# B&R Automation Studio project NAINV104C00R8L515F00 (part 22)

#### Local.var
```iecst
(*2019-06-17*)
(**)
(*Local Action, State & Status*)
VAR
	eAct : eConvAction := ConvActIdle;
	eStat : eConvAction := ConvActIdle;
	eStatus : eFBStatus := Idle;
	udiStatus : UDINT := 0;
	sStatTxt : STRING[200] := '';
	a_sStatText : ARRAY[0..60] OF STRING[200] := ['Idling','Initializing','Initializing With Reverse','Initializing With Pusher','Initializing With Puller','Initializing With Reject','Initializing With Inspection','Entering Board','Entering Board Until Inlet Signal Off','Entering Board With Reverse','Reversing Board','Reversing Board With Immediate Start Conv','Entering Board With Puller','Entering Board With Reject','Entering Board With Inspection','Pre Exiting Board','Resuming Reject Board',2('Exiting Board'),2('Exiting Board With Pusher'),'Pusher Setting All Control','Pusher Resetting All Control','Pusher Setting Extend','Pusher Setting Retract','Pusher Extending','Pusher Retracting','Puller Setting All Control','Puller Resetting All Control','Puller Setting Extend','Puller Setting Retract','Puller Extending','Puller Retracting','Rotating Setting All Control','Rotating Resetting All Control','Rotating Setting Home','Rotating Setting Remote','Rotating Turning Home','Rotating Turning Remote','Reject Setting All Control','Reject Resetting All Control','Reject Setting Up','Reject Setting Down','Reject Going Up','Reject Going Down','Stopping','Stopping With Pusher','Stopping With Puller','Stopping With Reject','Turning On Motor Signal','Turning On Motor Direction','Turning Off Motor Signal','Turning Off Motor Direction','Turning On All Motor Output','Turning Off All Motor Output',6('')];
END_VAR
(**)
(*Local Alarm*)
VAR
	tyAlmData : tyAlmDat;
	a_tyAlmText : ARRAY[10000..10199] OF tyAlmTxt := [(sAlmText:='Multi Board Detected While Conveyor Initial',sRcyText:='Operation Interrupted By Multiple Board. Remove Extra Boards And Resume Operation.'),(sAlmText:='Board Not Present At Outlet Sensor (L - R) While Conveyor Initial',sRcyText:='Operation Interrupted By Jam Board. Remove The Jam Board To Resume Operation.'),(sAlmText:='Board Not Present At Outlet Sensor (R - L) While Conveyor Initial',sRcyText:='Operation Interrupted By Jam Board. Remove The Jam Board To Resume Operation.'),(sAlmText:='Multi Board Detected While Conveyor Initial With Reverse',sRcyText:='Operation Interrupted By Multiple Board. Remove Extra Boards And Resume Operation.'),(sAlmText:='Board Not Present At Outlet Sensor (L - R) While Conveyor Initial With Reverse',sRcyText:='Operation Interrupted By Jam Board. Remove The Jam Board To Resume Operation.'),(sAlmText:='Board Not Present At Outlet Sensor (R - L) While Conveyor Initial With Reverse',sRcyText:='Operation Interrupted By Jam Board. Remove The Jam Board To Resume Operation.'),(sAlmText:='Pusher Extend Sensor Off Time Out In Retract Check While Conveyor Initial With Pusher',sRcyText:='Sensor Timeout Expired Before Operation Completed. Sensor Operation Is Abnormal. Solve The Error To Resume Operation.'),(sAlmText:='Pusher Retract Sensor On Time Out In Retract Check While Conveyor Initial With Pusher',sRcyText:='Sensor Timeout Expired Before Operation Completed. Sensor Operation Is Abnormal. Solve The Error To Resume Operation.'),(sAlmText:='Pusher Retract Safety Sensor Error In Retract Check While Conveyor Initial With Pusher',sRcyText:='Safety System Has Been Triggered. All Operations Are Disable. Remove the Obstacle That Triggered The Safety Interlock To Resume Operation.'),(sAlmText:='Multi Board Detected While Conveyor Initial With Pusher',sRcyText:='Operation Interrupted By Multiple Board. Remove Extra Boards And Resume Operation.'),(sAlmText:='Board Not Present At Outlet Sensor (L - R) While Conveyor Initial With Pusher',sRcyText:='Operation Interrupted By Jam Board. Remove The Jam Board To Resume Operation.'),(sAlmText:='Board Not Present At Outlet Sensor (R - L) While Conveyor Initial With Pusher',sRcyText:='Operation Interrupted By Jam Board. Remove The Jam Board To Resume Operation.'),(sAlmText:='Rotator Home Sensor On Time Out In Home Check While Conveyor Initial With Puller',sRcyText:='Sensor Timeout Expired Before Operation Completed. Sensor Operation Is Abnormal. Solve The Error To Resume Operation.'),(sAlmText:='Rotator Remote Sensor Off Time Out In Home Check While Conveyor Initial With Puller',sRcyText:='Sensor Timeout Expired Before Operation Completed. Sensor Operation Is Abnormal. Solve The Error To Resume Operation.'),(sAlmText:='Rotator Home Safety Sensor Error In Home Check While Conveyor Initial With Puller',sRcyText:='Safety System Has Been Triggered. All Operations Are Disable. Remove the Obstacle That Triggered The Safety Interlock To Resume Operation.'),(sAlmText:='Puller Extend Sensor Off Time Out In Retract Check While Conveyor Initial With Puller',sRcyText:='Sensor Timeout Expired Before Operation Completed. Sensor Operation Is Abnormal. Solve The Error To Resume Operation.'),(sAlmText:='Puller Retract Sensor On Time Out In Retract Check While Conveyor Initial With Puller',sRcyText:='Sensor Timeout Expired Before Operation Completed. Sensor Operation Is Abnormal. Solve The Error To Resume Operation.'),(sAlmText:='Puller Retract Safety Sensor Error In Retract Check While Conveyor Initial With Puller',sRcyText:='Safety System Has Been Triggered. All Operations Are Disable. Remove the Obstacle That Triggered The Safety Interlock To Resume Operation.'),(sAlmText:='Multi Board Detected While Conveyor Initial With Puller',sRcyText:='Operation Interrupted By Multiple Board. Remove Extra Boards And Resume Operation.'),(sAlmText:='Board Not Present At Outlet Sensor (L - R) While Conveyor Initial With Puller',sRcyText:='Operation Interrupted By Jam Board. Remove The Jam Board To Resume Operation.'),(sAlmText:='Board Not Present At Outlet Sensor (R - L) While Conveyor Initial With Puller',sRcyText:='Operation Interrupted By Jam Board. Remove The Jam Board To Resume Operation.'),(sAlmText:='Multi Board Detected While Conveyor Enter Board',sRcyText:='Operation Interrupted By Multiple Board. Remove Extra Boards And Resume Operation.'),(sAlmText:='Multi Board Detected While Conveyor Enter Board With Reverse',sRcyText:='Operation Interrupted By Multiple Board. Remove Extra Boards And Resume Operation.'),(sAlmText:='Puller Extend Sensor On Time Out In Extend Check While Conveyor Enter With Puller',sRcyText:='Sensor Timeout Expired Before Operation Completed. Sensor Operation Is Abnormal. Solve The Error To Resume Operation.'),(sAlmText:='Puller Retract Sensor Off Time Out In Extend Check While Conveyor Enter With Puller',sRcyText:='Sensor Timeout Expired Before Operation Completed. Sensor Operation Is Abnormal. Solve The Error To Resume Operation.'),(sAlmText:='Puller Extend Safety Sensor Error In Extend Check While Conveyor Enter With Puller',sRcyText:='Safety System Has Been Triggered. All Operations Are Disable. Remove the Obstacle That Triggered The Safety Interlock To Resume Operation.'),(sAlmText:='Rotator Home Sensor Off Time Out In Remote Check While Conveyor Enter With Puller',sRcyText:='Sensor Timeout Expired Before Operation Completed. Sensor Operation Is Abnormal. Solve The Error To Resume Operation.'),(sAlmText:='Rotator Remote Sensor On Time Out In Remote Check While Conveyor Enter With Puller',sRcyText:='Sensor Timeout Expired Before Operation Completed. Sensor Operation Is Abnormal. Solve The Error To Resume Operation.'),(sAlmText:='Rotator Remote Safety Sensor Error In Remote Check While Conveyor Enter With Puller',sRcyText:='Safety System Has Been Triggered. All Operations Are Disable. Remove the Obstacle That Triggered The Safety Interlock To Resume Operation.'),(sAlmText:='Puller Extend Sensor Off Time Out In Retract Check While Conveyor Enter With Puller',sRcyText:='Sensor Timeout Expired Before Operation Completed. Sensor Operation Is Abnormal. Solve The Error To Resume Operation.'),(sAlmText:='Puller Retract Sensor On Time Out In Retract Check While Conveyor Enter With Puller',sRcyText:='Sensor Timeout Expired Before Operation Completed. Sensor Operation Is Abnormal. Solve The Error To Resume Operation.'),(sAlmText:='Puller Retract Safety Sensor Error In Retract Check While Conveyor Enter With Puller',sRcyText:='Safety System Has Been Triggered. All Operations Are Disable. Remove the Obstacle That Triggered The Safety Interlock To Resume Operation.'),(sAlmText:='Rotator Home Sensor On Time Out In Home Check While Conveyor Enter With Puller',sRcyText:='Sensor Timeout Expired Before Operation Completed. Sensor Operation Is Abnormal. Solve The Error To Resume Operation.'),(sAlmText:='Rotator Remote Sensor Off Time Out In Home Check While Conveyor Enter With Puller',sRcyText:='Sensor Timeout Expired Before Operation Completed. Sensor Operation Is Abnormal. Solve The Error To Resume Operation.'),(sAlmText:='Rotator Home Safety Sensor Error In Home Check While Conveyor Enter With Puller',sRcyText:='Safety System Has Been Triggered. All Operations Are Disable. Remove the Obstacle That Triggered The Safety Interlock To Resume Operation.'),(sAlmText:='Multi Board Detected While Conveyor Enter With Puller',sRcyText:='Operation Interrupted By Multiple Board. Remove Extra Boards And Resume Operation.'),(sAlmText:='Multi Board Detected While Conveyor Pre-Exit Board',sRcyText:='Operation Interrupted By Multiple Board. Remove Extra Boards And Resume Operation.'),(sAlmText:='Board Missing While Conveyor Pre-Exit Board',sRcyText:='Operation Interrupted By Jam Board. Remove The Jam Board To Resume Operation.'),(sAlmText:='Multi Board Detected While Conveyor Exit Board',sRcyText:='Operation Interrupted By Multiple Board. Remove Extra Boards And Resume Operation.'),(sAlmText:='Multi Board Detected While Conveyor Exit Board With Pusher',sRcyText:='Operation Interrupted By Multiple Board. Remove Extra Boards And Resume Operation.'),(sAlmText:='Pusher Extend Sensor On Time Out In Extend Check While Conveyor Exit Board With Pusher',sRcyText:='Sensor Timeout Expired Before Operation Completed. Sensor Operation Is Abnormal. Solve The Error To Resume Operation.'),(sAlmText:='Pusher Retract Sensor Off Time Out In Extend Check While Conveyor Exit Board With Pusher',sRcyText:='Sensor Timeout Expired Before Operation Completed. Sensor Operation Is Abnormal. Solve The Error To Resume Operation.'),(sAlmText:='Pusher Extend Safety Sensor Error In Extend Check While Conveyor Exit Board With Pusher',sRcyText:='Safety System Has Been Triggered. All Operations Are Disable. Remove the Obstacle That Triggered The Safety Interlock To Resume Operation.'),(sAlmText:='Pusher Extend Sensor Off Time Out In Retract Check While Conveyor Exit Board With Pusher',sRcyText:='Sensor Timeout Expired Before Operation Completed. Sensor Operation Is Abnormal.Solve The Error To Resume Operation.'),(sAlmText:='Pusher Retract Sensor On Timeout In Retract Check While Conveyor Exit Board With Pusher',sRcyText:='Sensor Timeout Expired Before Operation Completed. Sensor Operation Is Abnormal. Solve The Error To Resume Operation.'),(sAlmText:='Pusher Retract Safety Sensor Error In Retract Check While Conveyor Exit Board With Pusher',sRcyText:='Safety System Has Been Triggered. All Operations Are Disable. Remove the Obstacle That Triggered The Safety Interlock To Resume Operation.'),(sAlmText:='Pusher Extend Sensor On Time Out In Extend Check While Pusher Extend',sRcyText:='Sensor Timeout Expired Before Operation Completed. Sensor Operation Is Abnormal. Solve The Error To Resume Operation.'),(sAlmText:='Pusher Retract Sensor Off Time Out In Extend Check While Pusher Extend',sRcyText:='Sensor Timeout Expired Before Operation Completed. Sensor Operation Is Abnormal. Solve The Error To Resume Operation.'),(sAlmText:='Pusher Extend Safety Sensor Error In Extend Check While Pusher Extend',sRcyText:='Safety System Has Been Triggered. All Operations Are Disable. Remove the Obstacle That Triggered The Safety Interlock To Resume Operation.'),(sAlmText:='Pusher Extend Sensor Off Time Out In Retract Check While Pusher Retract',sRcyText:='Sensor Timeout Expired Before Operation Completed. Sensor Operation Is Abnormal. Solve The Error To Resume Operation.'),(sAlmText:='Pusher Retract Sensor On Time Out In Retract Check While Pusher Retract',sRcyText:='Sensor Timeout Expired Before Operation Completed. Sensor Operation Is Abnormal. Solve The Error To Resume Operation.'),(sAlmText:='Pusher Retract Safety Sensor Error In Retract Check While Pusher Retract',sRcyText:='Safety System Has Been Triggered. All Operations Are Disable. Remove the Obstacle That Triggered The Safety Interlock To Resume Operation.'),(sAlmText:='Puller Extend Sensor On Time Out In Extend Check While Puller Extend',sRcyText:='Sensor Timeout Expired Before Operation Completed. Sensor Operation Is Abnormal. Solve The Error To Resume Operation.'),(sAlmText:='Puller Retract Sensor Off Time Out In Extend Check While Puller Extend',sRcyText:='Sensor Timeout Expired Before Operation Completed. Sensor Operation Is Abnormal. Solve The Error To Resume Operation.'),(sAlmText:='Puller Extend Safety Sensor Error In Extend Check While Puller Extend',sRcyText:='Safety System Has Been Triggered. All Operations Are Disable. Remove the Obstacle That Triggered The Safety Interlock To Resume Operation.'),(sAlmText:='Puller Extend Sensor Off Time Out In Retract Check While Puller Retract',sRcyText:='Sensor Timeout Expired Before Operation Completed. Sensor Operation Is Abnormal. Solve The Error To Resume Operation.'),(sAlmText:='Puller Retract Sensor On Time Out In Retract Check While Puller Retract',sRcyText:='Sensor Timeout Expired Before Operation Completed. Sensor Operation Is Abnormal. Solve The Error To Resume Operation.'),(sAlmText:='Puller Retract Safety Sensor Error In Retract Check While Puller Retract',sRcyText:='Safety System Has Been Triggered. All Operations Are Disable. Remove the Obstacle That Triggered The Safety Interlock To Resume Operation.'),(sAlmText:='Rotator Home Sensor On Time Out In Home Check While Rotator Home',sRcyText:='Sensor Timeout Expired Before Operation Completed. Sensor Operation Is Abnormal. Solve The Error To Resume Operation.'),(sAlmText:='Rotator Remote Sensor Off Time Out In Home Check While Rotator Home',sRcyText:='Sensor Timeout Expired Before Operation Completed. Sensor Operation Is Abnormal. Solve The Error To Resume Operation.'),(sAlmText:='Rotator Home Safety Sensor Error In Home Check While Rotator Home',sRcyText:='Safety System Has Been Triggered. All Operations Are Disable. Remove the Obstacle That Triggered The Safety Interlock To Resume Operation.'),(sAlmText:='Rotator Home Sensor Off Time Out In Remote Check While Rotator Remote',sRcyText:='Sensor Timeout Expired Before Operation Completed. Sensor Operation Is Abnormal. Solve The Error To Resume Operation.'),(sAlmText:='Rotator Remote Sensor On Time Out In Remote Check While Rotator Remote',sRcyText:='Sensor Timeout Expired Before Operation Completed. Sensor Operation Is Abnormal. Solve The Error To Resume Operation.'),(sAlmText:='Rotator Remote Safety Sensor Error In Remote Check While Rotator Remote',sRcyText:='Safety System Has Been Triggered. All Operations Are Disable. Remove the Obstacle That Triggered The Safety Interlock To Resume Operation.'),(sAlmText:='Pusher Extend Sensor Off Time Out In Retract Check While Stop With Pusher',sRcyText:='Sensor Timeout Expired Before Operation Completed. Sensor Operation Is Abnormal. Solve The Error To Resume Operation.'),(sAlmText:='Pusher Retract Sensor On Time Out In Retract Check While Stop With Pusher',sRcyText:='Sensor Timeout Expired Before Operation Completed. Sensor Operation Is Abnormal. Solve The Error To Resume Operation.'),(sAlmText:='Pusher Retract Safety Sensor Error In Retract Check While Stop With Pusher',sRcyText:='Safety System Has Been Triggered. All Operations Are Disable. Remove the Obstacle That Triggered The Safety Interlock To Resume Operation.'),(sAlmText:='Rotator Home Sensor On Time Out In Home Check While Stop With Puller',sRcyText:='Sensor Timeout Expired Before Operation Completed. Sensor Operation Is Abnormal. Solve The Error To Resume Operation.'),(sAlmText:='Rotator Remote Sensor Off Time Out In Home Check While Stop With Puller',sRcyText:='Sensor Timeout Expired Before Operation Completed. Sensor Operation Is Abnormal. Solve The Error To Resume Operation.'),(sAlmText:='Rotator Home Safety Sensor Error In Home Check While Stop With Puller',sRcyText:='Safety System Has Been Triggered. All Operations Are Disable. Remove the Obstacle That Triggered The Safety Interlock To Resume Operation.'),(sAlmText:='Puller Extend Sensor Off Time Out In Retract Check While Stop With Puller',sRcyText:='Sensor Timeout Expired Before Operation Completed. Sensor Operation Is Abnormal. Solve The Error To Resume Operation.'),(sAlmText:='Puller Retract Sensor On Time Out In Retract Check While Stop With Puller',sRcyText:='Sensor Timeout Expired Before Operation Completed. Sensor Operation Is Abnormal. Solve The Error To Resume Operation.'),(sAlmText:='Puller Retract Safety Sensor Error In Retract Check While Stop With Puller',sRcyText:='Safety System Has Been Triggered. All Operations Are Disable. Remove the Obstacle That Triggered The Safety Interlock To Resume Operation.'),(sAlmText:='Reject Up Sensor On Time Out In Up Check While Reject Up',sRcyText:='Sensor Timeout Expired Before Operation Completed. Sensor Operation Is Abnormal. Solve The Error To Resume Operation.'),(sAlmText:='Reject Down Sensor Off Time Out In Up Check While Reject Up',sRcyText:='Sensor Timeout Expired Before Operation Completed. Sensor Operation Is Abnormal. Solve The Error To Resume Operation.'),(sAlmText:='Reject Up Safety Sensor Error In Up Check While Reject Up',sRcyText:='Safety System Has Been Triggered. All Operations Are Disable. Remove the Obstacle That Triggered The Safety Interlock To Resume Operation.'),(sAlmText:='Reject Up Sensor Off Time Out In Down Check While Reject Down',sRcyText:='Sensor Timeout Expired Before Operation Completed. Sensor Operation Is Abnormal. Solve The Error To Resume Operation.'),(sAlmText:='Reject Down Sensor On Time Out In Down Check While Reject Down',sRcyText:='Sensor Timeout Expired Before Operation Completed. Sensor Operation Is Abnormal. Solve The Error To Resume Operation.'),(sAlmText:='Reject Down Safety Sensor Error In Down Check While Reject Down',sRcyText:='Safety System Has Been Triggered. All Operations Are Disable. Remove the Obstacle That Triggered The Safety Interlock To Resume Operation.'),(sAlmText:='Multi Board Detected While Conveyor Initial With Reject',sRcyText:='Operation Interrupted By Multiple Board. Remove Extra Boards And Resume Operation.'),(sAlmText:='Board Not Present At Outlet Or Middle Sensor (L - R) While Conveyor Initial With Reject',sRcyText:='Operation Interrupted By Jam Board. Remove The Jam Board To Resume Operation.'),(sAlmText:='Board Not Present At Outlet Or Middle Sensor (R - L) While Conveyor Initial With Reject',sRcyText:='Operation Interrupted By Jam Board. Remove The Jam Board To Resume Operation.'),(sAlmText:='Reject Up Sensor On Time Out In Up Check While Conveyor Initial With Reject',sRcyText:='Sensor Timeout Expired Before Operation Completed. Sensor Operation Is Abnormal. Solve The Error To Resume Operation.'),(sAlmText:='Reject Down Sensor Off Time Out In Up Check While Conveyor Initial With Reject',sRcyText:='Sensor Timeout Expired Before Operation Completed. Sensor Operation Is Abnormal. Solve The Error To Resume Operation.'),(sAlmText:='Reject Up Safety Sensor Error In Up Check While Conveyor Initial With Reject',sRcyText:='Safety System Has Been Triggered. All Operations Are Disable. Remove the Obstacle That Triggered The Safety Interlock To Resume Operation.'),(sAlmText:='Multi Board Detected While Conveyor Initial With Inspect',sRcyText:='Operation Interrupted By Multiple Board. Remove Extra Boards And Resume Operation.'),(sAlmText:='Board Not Present At Outlet Or Middle Sensor (L - R) While Conveyor Initial With Inspection',sRcyText:='Operation Interrupted By Jam Board. Remove The Jam Board To Resume Operation.'),(sAlmText:='Board Not Present At Outlet Or Middle Sensor (R - L) While Conveyor Initial With Inspection',sRcyText:='Operation Interrupted By Jam Board. Remove The Jam Board To Resume Operation.'),(sAlmText:='Reject Up Sensor On Time Out In Up Check While Conveyor Initial With Reject',sRcyText:='Sensor Timeout Expired Before Operation Completed. Sensor Operation Is Abnormal. Solve The Error To Resume Operation.'),(sAlmText:='Reject Down Sensor Off Time Out In Up Check While Conveyor Initial With Reject',sRcyText:='Sensor Timeout Expired Before Operation Completed. Sensor Operation Is Abnormal. Solve The Error To Resume Operation.'),(sAlmText:='Reject Up Safety Sensor Error In Up Check While Conveyor Initial With Reject',sRcyText:='Safety System Has Been Triggered. All Operations Are Disable. Remove the Obstacle That Triggered The Safety Interlock To Resume Operation.'),(sAlmText:='Multi Board Detected While Conveyor Initial With Reject',sRcyText:='Operation Interrupted By Multiple Board. Remove Extra Boards And Resume Operation.'),(sAlmText:='Board Not Present At Outlet Sensor (L - R) While Conveyor Initial With Reject',sRcyText:='Operation Interrupted By Jam Board. Remove The Jam Board To Resume Operation.'),(sAlmText:='Board Not Present At Outlet Sensor (R - L) While Conveyor Initial With Reject',sRcyText:='Operation Interrupted By Jam Board. Remove The Jam Board To Resume Operation.'),(sAlmText:='Multi Board Detected While Conveyor Entering With Reject',sRcyText:='Operation Interrupted By Multiple Board. Remove Extra Boards And Resume Operation.'),(sAlmText:='Reject Up Sensor On Time Out In Up Check While Conveyor Entering With Reject',sRcyText:='Sensor Timeout Expired Before Operation Completed. Sensor Operation Is Abnormal. Solve The Error To Resume Operation.'),(sAlmText:='Reject Down Sensor Off Time Out In Up Check While Conveyor Entering With Reject',sRcyText:='Sensor Timeout Expired Before Operation Completed. Sensor Operation Is Abnormal. Solve The Error To Resume Operation.'),(sAlmText:='Reject Up Safety Sensor Error In Up Check While Conveyor Entering With Reject',sRcyText:='Safety System Has Been Triggered. All Operations Are Disable. Remove the Obstacle That Triggered The Safety Interlock To Resume Operation.'),(sAlmText:='Multi Board Detected While Conveyor Entering With Inspection',sRcyText:='Operation Interrupted By Multiple Board. Remove Extra Boards And Resume Operation.'),(sAlmText:='Board Detect In Middle Sensor While Resuming Rejected Board',sRcyText:='Operation Interrupted By Jam Board. Remove The Jam Board To Resume Operation.'),(sAlmText:='Reject Up Sensor Off Time Out In Down Check While Resuming Rejected Board',sRcyText:='Sensor Timeout Expired Before Operation Completed. Sensor Operation Is Abnormal. Solve The Error To Resume Operation.'),(sAlmText:='Reject Down Sensor On Time Out In Down Check While Resuming Rejected Board',sRcyText:='Sensor Timeout Expired Before Operation Completed. Sensor Operation Is Abnormal. Solve The Error To Resume Operation.'),(sAlmText:='Reject Down Safety Sensor Error In Down Check While Resuming Rejected Board',sRcyText:='Safety System Has Been Triggered. All Operations Are Disable. Remove the Obstacle That Triggered The Safety Interlock To Resume Operation.'),(sAlmText:='Multi Board Detected While Resuming Rejected Board',sRcyText:='Operation Interrupted By Multiple Board. Remove Extra Boards And Resume Operation.'),(sAlmText:='Board Not Present At Outlet Sensor (L - R) While Resuming Rejected Board',sRcyText:='Operation Interrupted By Jam Board. Remove The Jam Board To Resume Operation.'),(sAlmText:='Board Not Present At Outlet Sensor (R - L) While Resuming Rejected Board',sRcyText:='Operation Interrupted By Jam Board. Remove The Jam Board To Resume Operation.'),(sAlmText:='Multi Board Detected While Conveyor Exit Board',sRcyText:='Operation Interrupted By Multiple Board. Remove Extra Boards And Resume Operation.'),(sAlmText:='Multi Board Detected While Conveyor Exit Board With Pusher',sRcyText:='Operation Interrupted By Multiple Board. Remove Extra Boards And Resume Operation.'),(sAlmText:='Pusher Extend Sensor On Time Out In Extend Check While Conveyor Exit Board With Pusher',sRcyText:='Sensor Timeout Expired Before Operation Completed. Sensor Operation Is Abnormal. Solve The Error To Resume Operation.'),(sAlmText:='Pusher Retract Sensor Off Time Out In Extend Check While Conveyor Exit Board With Pusher',sRcyText:='Sensor Timeout Expired Before Operation Completed. Sensor Operation Is Abnormal. Solve The Error To Resume Operation.'),(sAlmText:='Pusher Extend Safety Sensor Error In Extend Check While Conveyor Exit Board With Pusher',sRcyText:='Safety System Has Been Triggered. All Operations Are Disable. Remove the Obstacle That Triggered The Safety Interlock To Resume Operation.'),(sAlmText:='Pusher Extend Sensor Off Time Out In Retract Check While Conveyor Exit Board With Pusher',sRcyText:='Sensor Timeout Expired Before Operation Completed. Sensor Operation Is Abnormal. Solve The Error To Resume Operation.'),(sAlmText:='Pusher Retract Sensor On Time Out In Retract Check While Conveyor Exit Board With Pusher',sRcyText:='Sensor Timeout Expired Before Operation Completed. Sensor Operation Is Abnormal. Solve The Error To Resume Operation.'),(sAlmText:='Pusher Retract Safety Sensor Error In Retract Check While Conveyor Exit Board With Pusher',sRcyText:='Safety System Has Been Triggered. All Operations Are Disable. Remove the Obstacle That Triggered The Safety Interlock To Resume Operation.'),(sAlmText:='Transfer In Time Out While Conveyor Enter Board',sRcyText:='Timeout Expired Before Operation Completed. Transmission Abnormal. Remove the Obstacle (If Exists) To Resume Operation.'),(sAlmText:='Transfer In Time Out While Conveyor Enter Board With Reverse',sRcyText:='Timeout Expired Before Operation Completed. Transmission Abnormal. Remove the Obstacle (If Exists) To Resume Operation.'),(sAlmText:='Transfer In Time Out While Conveyor Enter With Puller',sRcyText:='Timeout Expired Before Operation Completed. Transmission Abnormal. Remove the Obstacle (If Exists) To Resume Operation.'),(sAlmText:='Transfer In Time Out While Conveyor Entering With Reject',sRcyText:='Timeout Expired Before Operation Completed. Transmission Abnormal. Remove the Obstacle (If Exists) To Resume Operation.'),(sAlmText:='Transfer In Time Out While Conveyor Entering With Inspection',sRcyText:='Timeout Expired Before Operation Completed. Transmission Abnormal. Remove the Obstacle (If Exists) To Resume Operation.'),(sAlmText:='Transfer Out Time Out While Conveyor Exit Board',sRcyText:='Timeout Expired Before Operation Completed. Transmission Abnormal. Remove the Obstacle (If Exists) To Resume Operation.'),(sAlmText:='Transfer Out Time Out While Conveyor Exit Board With Pusher',sRcyText:='Timeout Expired Before Operation Completed. Transmission Abnormal. Remove the Obstacle (If Exists) To Resume Operation.'),(sAlmText:='Transfer Out Time Out While Conveyor Exit Board',sRcyText:='Timeout Expired Before Operation Completed. Transmission Abnormal. Remove the Obstacle (If Exists) To Resume Operation.'),(sAlmText:='Transfer Out Time Out While Conveyor Exit Board With Pusher',sRcyText:='Timeout Expired Before Operation Completed. Transmission Abnormal. Remove the Obstacle (If Exists) To Resume Operation.'),(sAlmText:='Multi Board Detected While Conveyor Enter Board To Inlet Off',sRcyText:='Operation Interrupted By Multiple Board. Remove Extra Boards And Resume Operation.'),(sAlmText:='Transfer In Time Out While Conveyor Enter Board To Inlet Off',sRcyText:='Timeout Expired Before Operation Completed. Transmission Abnormal. Remove the Obstacle (If Exists) To Resume Operation.'),(sAlmText:='Transfer In Time Out While Conveyor Reversing Board',sRcyText:='Timeout Expired Before Operation Completed. Transmission Abnormal. Remove the Obstacle (If Exists) To Resume Operation.'),0,73((0))];
END_VAR
(**)
(*Local Output*)
VAR
	bHvBrd : BOOL;
	bRejHvBrd : BOOL;
	bInspHvBrd : BOOL;
	bGdBrd : BOOL;
	bLmtSenActivated : BOOL;
	bMtrSigOnOrLToR : BOOL;
	bMtrDirOrRToL : BOOL;
	bPshrExtCtrl : BOOL;
	bPshrTwoOutputControl : BOOL := FALSE;
	bPshrExtended : BOOL;
	bPshrRetracted : BOOL;
	bPullerExtCtrl : BOOL;
	bPullerRetCtrl : BOOL;
	bPullerTwoOutputControl : BOOL := TRUE;
	bPullerExtended : BOOL;
	bPullerRetracted : BOOL;
	bRotRemoteCtrl : BOOL;
	bRotTwoOutputControl : BOOL := FALSE;
	bRotAtRemote : BOOL;
	bRotAtHome : BOOL;
	bRejectUpCtrl : BOOL;
	bRejectDownCtrl : BOOL;
	bRejectTwoOutputControl : BOOL := TRUE;
	bRejectAtUp : BOOL;
	bRejectAtDown : BOOL;
END_VAR
(**)
(*Local Input*)
VAR
	udiRstErr : UDINT := 0;
	bPrep : BOOL := TRUE;
	bEn : BOOL := TRUE;
	bDis : BOOL := FALSE;
	bManual : BOOL := FALSE;
	bLongBrdPrep : BOOL := FALSE;
	bLongBrdEn : BOOL := FALSE;
	bOnDirMod : BOOL := FALSE;
	diInitTm : DINT := 10000;
	diRevDlyTm : DINT := 500;
	tMtrOffDlyTm : TIME := T#0S;
	diTxInTimeOut : DINT := 10000;
	diTxOutTimeOut : DINT := 10000;
	eDirection : eConvDir := ConvDirLToR;
	bGdBrdInit : BOOL := TRUE;
	bGdBrdEnt : BOOL := TRUE;
	bLeftSen : BOOL := FALSE;
	bRightSen : BOOL := FALSE;
	bMiddleSen : BOOL := FALSE;
	bPullerChkSen : BOOL := FALSE;
	bPshrExtSen : BOOL := FALSE;
	bPshrRetSen : BOOL := FALSE;
	bPshrExtSafetySen : BOOL := TRUE;
	bPshrRetSafetySen : BOOL := TRUE;
	bPullerExtSen : BOOL := FALSE;
	bPullerRetSen : BOOL := FALSE;
	bPullerExtSafetySen : BOOL := TRUE;
	bPullerRetSafetySen : BOOL := TRUE;
	bRotHomeSen : BOOL := FALSE;
	bRotRemoteSen : BOOL := FALSE;
	bRotHomeSafetySen : BOOL := TRUE;
	bRotRemoteSafetySen : BOOL := TRUE;
	bRejectUpSen : BOOL := FALSE;
	bRejectDownSen : BOOL := FALSE;
	bRejectUpSafetySen : BOOL := TRUE;
	bRejectDownSafetySen : BOOL := TRUE;
	sProgNm : STRING[15] := 'Conv';
	tPshrExtTO : TIME := T#20s;
	tPshrRetTO : TIME := T#20s;
	tPullerExtTO : TIME := T#20s;
	tPullerRetTO : TIME := T#20s;
	tRotHomeTO : TIME := T#20s;
	tRotRemoteTO : TIME := T#20s;
	tRejectUpTO : TIME := T#20s;
	tRejectDownTO : TIME := T#20s;
	bNtSettingsLoadDone : BOOL := TRUE;
END_VAR
(**)
(*Local*)
VAR
	bRstErr : BOOL;
	udiRstErrOld : UDINT;
	bInitDone : BOOL;
	bInitialDone : BOOL;
	usiStep : USINT;
	bInletOff : BOOL;
	fbWaitTm : TON := (PT:=T#1s);
	eStatOld : eConvAction := ConvActIdle;
	fbInit : fbConvSenToSenTm;
	fbEnt : fbConvSenToSen;
	fbRev : fbConvSenToSenTm1;
	fbPreExit : fbConvSenToSenTm;
	fbExit : fbConvSenToSenOff;
	fbExit1 : fbConvSenToSenOff1;
	fbLongBrd : fbConvLongBrd;
	fbStop : fbConvMtrOff;
	fbPshrExtChk : fbPneuExtRetSenExtChk;
	fbPshrRetChk : fbPneuExtRetSenRetChk;
	fbPullerExtChk : fbPneuExtRetSenExtChk;
	fbPullerRetChk : fbPneuExtRetSenRetChk;
	fbRotHomeChk : fbPneuExtRetSenExtChk;
	fbRotRemoteChk : fbPneuExtRetSenRetChk;
	fbRejectUpChk : fbPneuExtRetSenExtChk;
	fbRejectDownChk : fbPneuExtRetSenRetChk;
	udiModuleNum : UDINT := 1501;
END_VAR
```

#### Act_Action.st
```iecst
(** 2019-03-25 **)
ACTION Act_Action:

	//Reset Error
	IF (eStatus = Error) AND bRstErr THEN
		p_eAct	:= ConvActIdle;
		eStat	:= ConvActIdle;
	END_IF

	//Set p_eAct
	IF eStatus = Idle OR eStatus = Busy OR eStatus = Done THEN
		eStat	:= p_eAct;
	END_IF

END_ACTION
```

#### Act_Alarm.st
```iecst
(** 2022-12-20 **)
ACTION Act_Alarm:

	//Error
	IF EDGEPOS(eStatus = Error) THEN

		tyAlmData.sProgNm		:= p_sProgNm;
		tyAlmData.udiCode		:= udiStatus;
		tyAlmData.eSeverity		:= AlmSeverityError;
		tyAlmData.udiRunTime	:= tyAlmData.udiRunTime + 1;
		tyAlmData.bAlm			:= TRUE;
		tyAlmData.udiModuleNum  := udiModuleNum;
		g_sConvProgNm		    := p_sProgNm;

		//Get Error Message
		IF tyAlmData.udiCode < 10000 OR tyAlmData.udiCode > 10199 THEN
			tyAlmData.sAlmMsg	:= 'Unknown';
			tyAlmData.sRcyMsg	:= 'Unknown';
		ELSE
			tyAlmData.sAlmMsg	:= a_tyAlmText[tyAlmData.udiCode].sAlmText;
			tyAlmData.sRcyMsg	:= a_tyAlmText[tyAlmData.udiCode].sRcyText;
		END_IF

		sStatTxt	:= tyAlmData.sAlmMsg;

	ELSIF bRstErr AND (tyAlmData.udiCode <> 0) THEN

		tyAlmData.udiCode	:= 0;
		tyAlmData.eSeverity	:= AlmSeverityNA;
		tyAlmData.sAlmMsg	:= '';
		tyAlmData.sRcyMsg	:= '';
		tyAlmData.bAlm		:= FALSE;
		sStatTxt	:= a_sStatText[eStat];

	END_IF

END_ACTION
```

#### Act_Background.st
```iecst
(** 2019-01-18 **)
ACTION Act_Background:

	IF p_bPshrExtSen = FALSE THEN
		bPshrExtended	:= FALSE;
	END_IF

	IF p_bPshrRetSen = FALSE THEN
		bPshrRetracted	:= FALSE;
	END_IF

	IF p_bPullerExtSen = FALSE THEN
		bPullerExtended	:= FALSE;
	END_IF

	IF p_bPullerRetSen = FALSE THEN
		bPullerRetracted	:= FALSE;
	END_IF

	IF p_bRotHomeSen = FALSE THEN
		bRotAtHome	:= FALSE;
	END_IF

	IF p_bRotRemoteSen = FALSE THEN
		bRotAtRemote	:= FALSE;
	END_IF

	IF p_bRejectUpSen = FALSE THEN
		bRejectAtUp	:= FALSE;
	END_IF

	IF p_bRejectDownSen = FALSE THEN
		bRejectAtDown	:= FALSE;
	END_IF

END_ACTION
```

#### Act_InitGlobal.st
```iecst
(** 2019-04-09 **)
ACTION Act_InitGlobal:

	(* Always Change If Project Change *)

	//Pass Data To Link
	p_bLinkOpsRun ACCESS p_OpsRun;
	p_bLinkOpsSimu ACCESS p_SimuRun;

	p_bLinkUIBypsInitConv ACCESS p_UIOpsBypsInitConv;
	p_eLinkMcParamUSCommMod ACCESS p_McParamUSCommMod;
	p_bLinkOpsInvertBrdInserted ACCESS p_OpsInvertBrdInserted;
	p_eLinkMcParamUSComm2Mod ACCESS p_McParamUSComm2Mod;
	p_bLinkOpsInvertOnceTwicePCBOut ACCESS p_OpsInvertOnceTwicePCBOut;
	p_usiLinkMcMod ACCESS p_ProdRcpCurrRcp0McMod;

	p_tyNtParamCurr ACCESS p_NtParamCurr;

	//Pass Data To Internal Use
	p_udiRstErr ACCESS p_RstErrReset;
	p_bManual ACCESS p_UIMnlMod;
	p_bOnDirMod ACCESS p_NtParamConvOnDirMod;
	p_diInitTm ACCESS p_McParamConvInitTm;
	p_diRevDlyTm ACCESS p_NtParamConvRevDlyTm;
	p_tMtrOffDlyTm ACCESS p_NtParamConvMtrOffDlyTm;
	p_diTxInTimeOut ACCESS p_McParamTranInErrDlyTm;
	p_diTxOutTimeOut ACCESS p_McParamTranOutErrDlyTm;
//	p_eDirection ACCESS p_NtParamProjConvDir;
	p_sProgNm ACCESS p_NtParamConvProgNm;
	p_bLeftSen ACCESS p_DIConvLftSen;
	p_bRightSen	ACCESS p_DIConvRgtSen;
	p_bNtSettingsLoadDone ACCESS p_StartupNtSettingsLoadDone;

	(* Always Change If Project Change *)

	//Routing
	p_bUSHermesDSRdy ACCESS p_USHermesDSRdy;
	p_bDSHermesUSRdy ACCESS  p_DSHermesUSRdy;
	p_bUSHermesReversalDSRdy ACCESS p_USHermes2DSRdy;
	p_bDSHermesReversalUSRdy ACCESS  p_DSHermes2USRdy;
END_ACTION
```

#### Act_Initial.st
```iecst
(** 2019-03-22 **)
ACTION Act_Initial:

	//Initial
	sStatTxt	:= a_sStatText[eStat];

	fbWaitTm(IN := FALSE);

	fbInit.bOnDirMod	:= p_bOnDirMod;
	fbInit.bStartSen	:= TRUE;
	fbInit.tMtrOffDlyTm	:= p_tMtrOffDlyTm;
	fbInit(bEn := FALSE);

	fbEnt.bOnDirMod		:= p_bOnDirMod;
	fbEnt.bStartSen		:= TRUE;
	fbEnt.tMtrOffDlyTm	:= p_tMtrOffDlyTm;
	fbEnt(bEn := FALSE);

	fbRev.bOnDirMod		:= p_bOnDirMod;
	fbRev.tTxDlyTm		:= DINT_TO_TIME(p_diRevDlyTm);
	fbRev.tMtrOffDlyTm	:= p_tMtrOffDlyTm;
	fbRev(bEn := FALSE);

	fbPreExit.bOnDirMod		:= p_bOnDirMod;
	fbPreExit.bStartSen		:= TRUE;
	fbPreExit.tMtrOffDlyTm	:= p_tMtrOffDlyTm;
	fbPreExit(bEn := FALSE);

	fbExit.bOnDirMod	:= p_bOnDirMod;
	fbExit.bStartSen	:= TRUE;
	fbExit.tMtrOffDlyTm	:= p_tMtrOffDlyTm;
	fbExit(bEn := FALSE);

	fbExit1.bOnDirMod		:= p_bOnDirMod;
	fbExit1.bStartSen		:= TRUE;
	fbExit1.tMtrOffDlyTm	:= p_tMtrOffDlyTm;
	fbExit1(bEn := FALSE);

	fbStop(bEn := FALSE);

	fbPshrExtChk.tTimeOut	:= p_tPshrExtTO;
	fbPshrExtChk(bEn := FALSE);

	fbPshrRetChk.tTimeOut	:= p_tPshrRetTO;
	fbPshrRetChk(bEn := FALSE);

	fbPullerExtChk.tTimeOut	:= p_tPullerExtTO;
	fbPullerExtChk(bEn := FALSE);

	fbPullerRetChk.tTimeOut	:= p_tPullerRetTO;
	fbPullerRetChk(bEn := FALSE);

	fbRotHomeChk.tTimeOut	:= p_tRotHomeTO;
	fbRotHomeChk(bEn := FALSE);

	fbRotRemoteChk.tTimeOut	:= p_tRotRemoteTO;
	fbRotRemoteChk(bEn := FALSE);

	fbRejectUpChk.tTimeOut	:= p_tRejectUpTO;
	fbRejectUpChk(bEn := FALSE);

	fbRejectDownChk.tTimeOut	:= p_tRejectDownTO;
	fbRejectDownChk(bEn := FALSE);

END_ACTION
```

#### Act_InitLocal.st
```iecst
(** 2019-03-25 **)
ACTION Act_InitLocal:

	//Input Reference Link To Local Variable
	p_eAct ACCESS ADR(eAct);
	p_udiRstErr ACCESS ADR(udiRstErr);
	p_bPrep ACCESS ADR(bPrep);
	p_bEn ACCESS ADR(bEn);
	p_bDis ACCESS ADR(bDis);

	p_bManual ACCESS ADR(bManual);
	p_bLongBrdPrep ACCESS ADR(bLongBrdPrep);
	p_bLongBrdEn ACCESS ADR(bLongBrdEn);
	p_bOnDirMod ACCESS ADR(bOnDirMod);
	p_diInitTm ACCESS ADR(diInitTm);
	p_diRevDlyTm ACCESS ADR(diRevDlyTm);
	p_tMtrOffDlyTm ACCESS ADR(tMtrOffDlyTm);
	p_diTxInTimeOut ACCESS ADR(diTxInTimeOut);
	p_diTxOutTimeOut ACCESS ADR(diTxOutTimeOut);
	p_eDirection ACCESS ADR(eDirection);
	p_bGdBrdEnt ACCESS ADR(bGdBrdEnt);
	p_bGdBrdInit ACCESS ADR(bGdBrdInit);
	p_sProgNm ACCESS ADR(sProgNm);
	p_tPshrExtTO ACCESS ADR(tPshrExtTO);
	p_tPshrRetTO ACCESS ADR(tPshrRetTO);
	p_tPullerExtTO ACCESS ADR(tPullerExtTO);
	p_tPullerRetTO ACCESS ADR(tPullerRetTO);
	p_tRotHomeTO ACCESS ADR(tRotHomeTO);
	p_tRotRemoteTO ACCESS ADR(tRotRemoteTO);
	p_tRejectUpTO ACCESS ADR(tRejectUpTO);
	p_tRejectDownTO ACCESS ADR(tRejectDownTO);
	p_bNtSettingsLoadDone ACCESS ADR(bNtSettingsLoadDone);

	p_bLeftSen ACCESS ADR(bLeftSen);
	p_bRightSen ACCESS ADR(bRightSen);
	p_bMiddleSen ACCESS ADR(bMiddleSen);
	p_bPullerChkSen ACCESS ADR(bPullerChkSen);
	p_bPshrExtSen ACCESS ADR(bPshrExtSen);
	p_bPshrRetSen ACCESS ADR(bPshrRetSen);
	p_bPshrExtSafetySen ACCESS ADR(bPshrExtSafetySen);
	p_bPshrRetSafetySen ACCESS ADR(bPshrRetSafetySen);
	p_bPullerExtSen ACCESS ADR(bPullerExtSen);
	p_bPullerRetSen ACCESS ADR(bPullerRetSen);
	p_bPullerExtSafetySen ACCESS ADR(bPullerExtSafetySen);
	p_bPullerRetSafetySen ACCESS ADR(bPullerRetSafetySen);
	p_bRotHomeSen ACCESS ADR(bRotHomeSen);
	p_bRotRemoteSen ACCESS ADR(bRotRemoteSen);
	p_bRotHomeSafetySen ACCESS ADR(bRotHomeSafetySen);
	p_bRotRemoteSafetySen ACCESS ADR(bRotRemoteSafetySen);
	p_bRejectUpSen ACCESS ADR(bRejectUpSen);
	p_bRejectDownSen ACCESS ADR(bRejectDownSen);
	p_bRejectUpSafetySen ACCESS ADR(bRejectUpSafetySen);
	p_bRejectDownSafetySen ACCESS ADR(bRejectDownSafetySen);

END_ACTION
```

#### Act_Link.st
```iecst
(** 2019-03-29 **)
ACTION Act_Link:

	IF p_bLinkUIBypsInitConv THEN
		p_diInitTm ACCESS ADR(diInitTm);
	ELSE
		p_diInitTm ACCESS p_McParamConvInitTm;
	END_IF

	IF EDGEPOS(eStatus = Error) THEN
		bMtrSigOnOrLToR	:= FALSE;
		bMtrDirOrRToL	:= FALSE;
	END_IF

	//Update Good/Bad Board
	IF p_eLinkMcParamUSCommMod = McSetCommModSMEMA THEN
		IF p_bLinkOpsInvertBrdInserted = TRUE THEN
			p_bGdBrdEnt	:= TRUE;
		ELSE
			p_bGdBrdEnt ACCESS p_USSMEMAUSGdBrdRdy;
		END_IF
	ELSIF p_eLinkMcParamUSCommMod = McSetCommModHermes THEN
		IF p_bLinkOpsInvertBrdInserted = TRUE THEN
			p_bGdBrdEnt	:= TRUE;
		ELSE
			p_bGdBrdEnt ACCESS p_USHermesUSGdRdy;
		END_IF
	END_IF

	IF p_eLinkMcParamUSComm2Mod = McSetCommModSMEMA THEN
		IF p_bLinkOpsInvertBrdInserted = TRUE THEN
			p_bGdBrdEnt := TRUE;
		ELSE
			p_bGdBrdEnt ACCESS p_USSMEMA2USGdBrdRdy;
		END_IF
	ELSIF p_eLinkMcParamUSComm2Mod = McSetCommModHermes THEN
		IF p_bLinkOpsInvertBrdInserted = TRUE THEN
			p_bGdBrdEnt	:= TRUE;
		ELSE
			p_bGdBrdEnt ACCESS p_USHermesUSGdRdy;
		END_IF
	END_IF

	//Reverse timeout
	fbRev.tTimeOut:= DINT_TO_TIME(p_diTxInTimeOut);

	//Conveyor Direction
	IF (p_usiLinkMcMod = 0 OR p_usiLinkMcMod = 1) OR ((p_usiLinkMcMod = 2 OR p_usiLinkMcMod = 3) AND NOT(p_bLinkOpsInvertOnceTwicePCBOut))   THEN
		p_eDirection ACCESS p_NtParamProjConvDir;
	ELSIF (p_usiLinkMcMod = 2 OR p_usiLinkMcMod = 3) AND p_bLinkOpsInvertOnceTwicePCBOut THEN
		p_eDirection ACCESS p_NtParamProjRtrnBrdConvDir;
	ELSIF p_usiLinkMcMod =4   THEN//USReversalRdy or DSReversalRdy
		IF EDGEPOS(p_bUSHermesReversalDSRdy OR p_bDSHermesReversalUSRdy) THEN
			p_eDirection ACCESS p_NtParamProjRtrnBrdConvDir;
		ELSIF  EDGEPOS(p_bUSHermesDSRdy OR p_bDSHermesUSRdy) THEN
			p_eDirection ACCESS p_NtParamProjConvDir;
		END_IF
	END_IF

END_ACTION
```

#### Act_LinkAction.st
```iecst
(** 2019-04-09 **)
ACTION Act_LinkAction:

	IF p_bLinkOpsRun = TRUE THEN
		p_eAct ACCESS p_OpsInvertConvAct;
	ELSIF p_bManual = TRUE THEN
		p_eAct ACCESS p_UIConvAct;
	ELSIF p_bLinkOpsSimu = TRUE THEN
		p_eAct ACCESS p_SimuInvConvAct;

	ELSE
		p_eAct ACCESS ADR(eAct);
	END_IF

END_ACTION
```

#### Act_LinkEn.st
```iecst
(** 2019-01-11 **)
ACTION Act_LinkEn:

	//Link bPrep, bEn & bDis

END_ACTION
```
